(* CoDeSys 2.3.9.37 project: Cap3_6.pro *)
(* Libraries: Standard.LIB 4.10.05 12:14:46 *)

(* Global variable list: Global_Variables *)
VAR_GLOBAL

(* Entradas *)
     A:BOOL;
     B:BOOL;
     Encendido:BOOL;

(*Salidas *)
  Bomba:BOOL;

END_VAR

(* Data type *)
TYPE
  Color :(rojo,verde,amarillo);
END_TYPE

(* Data type *)
TYPE MiEstructura :
   STRUCT
      Valor : INT;
      Med1 : INT;
      Luz : Color;
END_STRUCT
END_TYPE

(* POU PLC_PRG, ST *)
PROGRAM PLC_PRG
VAR
  posy:INT;
 Desague: BOOL;
END_VAR
Control();


IF Bomba=TRUE THEN
IF posy>-187 THEN
  posy:=posy-1;
END_IF
END_IF

IF Bomba=FALSE THEN
IF posy<52 THEN
  posy:=posy+1;
END_IF
END_IF



IF Desague=1 THEN
IF posy<48 THEN
posy:=posy+4;
END_IF
END_IF

IF posy<-121 THEN
  A:=TRUE;
ELSE
  A:=FALSE;
END_IF

IF posy<=-164 THEN
  B:=TRUE;
ELSE
  B:=FALSE;
END_IF
END_PROGRAM

(* POU Control, LD *)
PROGRAM Control
VAR

END_VAR
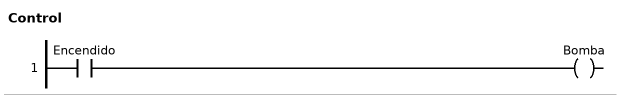
_LD_ (* Ladder Diagram *)
NETWORK 1
	[Encendido] --- (Bomba)
_END_LD_
(* the same logic as Structured Text *)
(* Network 1 *)
Bomba := Encendido;
END_PROGRAM

(* Visualisation Deposito
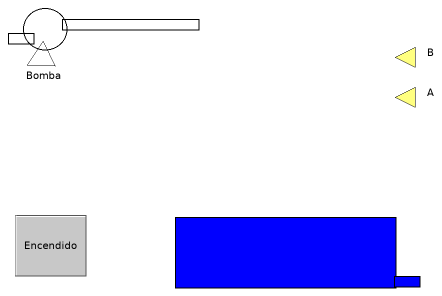
button at (60,228)-(131,289): text "Encendido"; toggles .Encendido
polygon at (440,60)-(460,80): alarm colour if .B; toggles .B
polygon at (440,100)-(460,120): alarm colour if .A; toggles .A
rectangle at (220,230)-(441,301): top PLC_PRG.posy
rectangle at (460,90)-(491,121): text "A"
rectangle at (460,50)-(491,81): text "B"
rectangle at (107,32)-(244,43): alarm colour if Bomba
ellipse at (68,21)-(112,63): alarm colour if Bomba
polygon at (72,54)-(100,79): alarm colour if Bomba
rectangle at (53,46)-(79,57): alarm colour if Bomba
rectangle at (59,74)-(118,103): text "Bomba"
2 more shapes without text or variables
1 elements of other kinds (tables, trends, ...) not read
*)
